TYPE ST_PositioningLaser_HWI :
STRUCT
  udiDistanceRaw          : UDINT;  
END_STRUCT
END_TYPE

(* stored: Version 1.1.0.1, ProductVersion 3.1.4024.12
   DUT ST_PositioningLaser_HWI: Id {ce224bb7-ae30-4d36-9efe-671c1e7ff197} *)
